(* IEC 61131-3 sources: Industry-PLC-LLM/data/PLCBEAD_repo/PLCBEAD_PLCEmbed-main/PLC-BEAD/Source/GEB/TOD_TO_REAL, 1 file *)

(* ---- TOD_TO_REAL.ST ---- *)
FUNCTION TOD_TO_REAL2:REAL
	VAR_INPUT
		IN :	UDINT;
	END_VAR
	TOD_TO_REAL2 := UDINT_TO_REAL(IN);
END_FUNCTION

PROGRAM program0
  VAR
	IN :	UDINT;
    CEIL5_OUT : REAL;
  END_VAR

  CEIL5_OUT := TOD_TO_REAL2(IN);
END_PROGRAM
